// TIA Portal V18 export
DATA_BLOCK "DevTestBlock"   // DB47
{ S7_Optimized_Access := 'FALSE' }
VERSION : 0.1
// stored: AutoNumber true, DBAccessibleFromOPCUA true, IsOnlyStoredInLoadMemory false, IsWriteProtectedInAS false
   VAR
      EnableAxisTest : Bool;
      Z2Halt : Bool;
      Z1Halt : Bool;
      XHalt : Bool;
      YHalt : Bool;
      GlobalHalt : Bool;
      TaskZ2E : Bool;
      TaskZ1M : Bool;
      TaskZ2M : Bool;
      TaskXM { S7_SetPoint := 'True'} : Bool;
      TaskYM : Bool;
      TestResetCommand : Bool;
      TestResetZ1 : Bool;
      TestResetZ2 : Bool;
      TestResetX : Bool;
      TestResetY : Bool;
      DoorSensor : Bool := true;   // True for testing to disable door sensors
      "Weight Test value" : UInt;
      DoorSensorPrintboxSkip : Bool := true;
      DoorSensor_Side : Bool := false;
      DoorSensor_PrintBox : Bool;
      AXIS_ackerror : Bool;
      AXIS_X_enable : Bool;
      AXIS_Y_enable : Bool;
      AXIS_Z1_enable : Bool;
      AXIS_jog1 : Bool := false;
      AXIS_jog2 : Bool;
      AXIS_X_velocity : Real;
      AXIS_X_position : Int;
      AXIS_execute : Bool;
      ConfigEPos : DWord := 16#0000_000F;
      "AXIS Warning" : Bool := false;
      "AXIS Error Fault" : Bool := false;
      "AXIS Enabled" : Bool := false;
      "AXIS Ready" : Bool := false;
      PurgeX : DInt := 480000;
      PurgeY : DInt := 90000;
      PurgeVelocity : DInt := 300;
      PurgeMove : Bool;
      "OLD off" : Bool;
      LED1 : Bool;
      LED2 : Bool;
      CappingHoming : Bool;
      reset : Bool;
      DamagedDoorSensorTemp : Bool := false;
      CappingEnable : Bool;
      TestYvelocity : DInt := 100000;
      TestingCappingStation : Bool;
      TestCapping01 : Bool;
      TestCapping02 : Bool;
      TestCapping03 : Bool;
      TestCappingNotUsed : Bool;
      ResetCounters : Bool;
      RET_VAL : Int;
      WebServerTest : Int := 1;
   END_VAR
BEGIN
END_DATA_BLOCK
